{attribute 'GeneratedUsingTerminal: EM7004-0000-0017'}
{attribute addProperty BoxType "EM7004-0000-0017"}
{attribute addProperty Id "Enable_PLSBOOL1"}
{attribute addProperty CRC "398073794"}
{attribute addProperty Size "1"}
TYPE Control_17BA1FC2 :
STRUCT
	{attribute addProperty Name "Enable_PLS"}
	Enable_PLS : BOOL;
END_STRUCT
END_TYPE

(* stored: Version 1.2.0.0, ProductVersion 3.1.4024.9
   DUT Control_17BA1FC2: Id {28316c46-87d3-493b-af8f-1b8632012bf4} *)
